(* PLC project Unnamed, Unknown Unnamed 1 *)
(* stored: creationDateTime 2023-03-10T10:37:17, modificationDateTime 2023-03-15T15:56:42 *)

(* ISBN 978-3-8348-0266-8, Lernaufgabe 2.1 *)
FUNCTION_BLOCK Silo_Valve_Control_System
  VAR_INPUT
    IN1 : BOOL;
    IN2 : BOOL;
    IN3 : BOOL;
    IN4 : BOOL;
  END_VAR
  VAR_OUTPUT
    OUT1 : BOOL;
  END_VAR

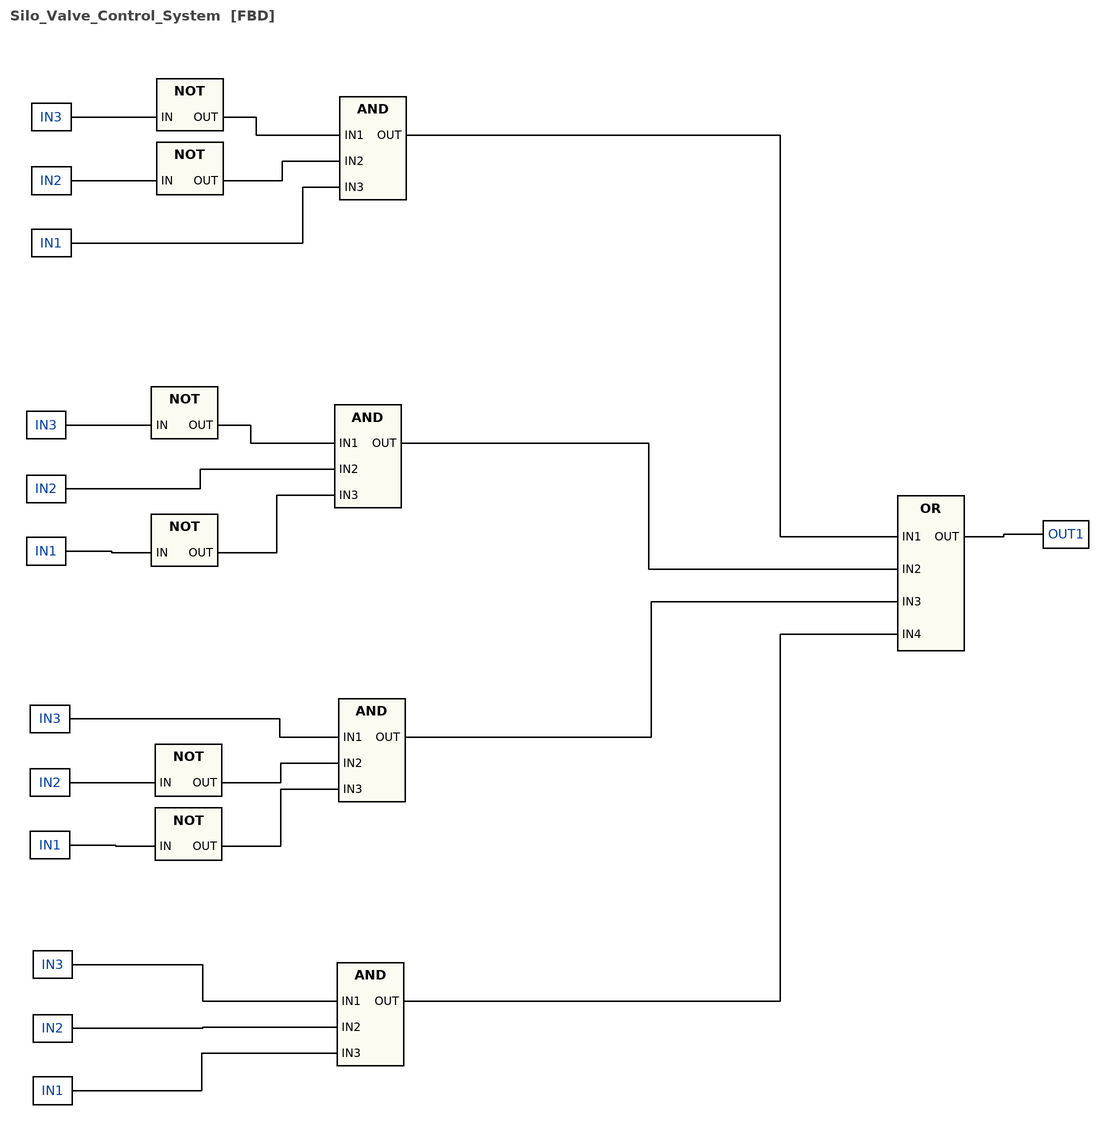
(* FBD diagram, written out as Structured Text *)
OUT1 := NOT IN3 AND NOT IN2 AND IN1 OR NOT IN3 AND IN2 AND NOT IN1 OR IN3 AND NOT IN2 AND NOT IN1 OR IN3 AND IN2 AND IN1;
END_FUNCTION_BLOCK

CONFIGURATION config
  RESOURCE resource1 ON PLC
  END_RESOURCE
END_CONFIGURATION
